// TIA Portal project "VISU_Registerlager_Template" (V14)

(* hardware
DEVICE "S7300/ET200M-Station_1"  S7-300 station
   slot 0: "Profilschiene_0"  Rail  6ES7 390-1***0-0AA0
   slot 2: "PLC_1"  CPU 315-2 PN/DP  6ES7 315-2EH13-0AB0  V2.6
      slot 1: "MPI/DP-Schnittstelle_1"  X1
      slot 2: "PROFINET-Schnittstelle_1"  PN-IO
         slot 1: "Port_1"  Port
*)

// ===== PLC "PLC_1"  CPU 315-2 PN/DP =====

VAR_GLOBAL   // PLC tag table "Standard-Variablentabelle"
   "CHAIN_REGISTER" AT %I10.0 : Bool;   // Förderkette Registerlager
   "REGISTER_ENGAGED" AT %I10.1 : Bool;   // Registerlager belegt
   "BELT_ENGAGED" AT %I10.2 : Bool;   // Förderband belegt
   "READ_SENSOR1" AT %I10.3 : Bool;   // Lesestation Sensor 1
   "READ_SENSOR2" AT %I10.4 : Bool;   // Lesestation Sensor 2
   "CONTROL_KEY" AT %I10.5 : Bool;   // Bedientaster
   "CHAIN_ON" AT %Q4.0 : Bool;   // Förderkette Regtisterlager an
   "LED_ON" AT %Q4.2 : Bool;   // LED an
   "BOX_NO" AT %MD1000 : DInt;   // Box-Nummer
   "BELT_ON" AT %Q4.1 : Bool;   // Förderband an
   "Merker TOF aktiv" AT %M0.0 : Bool;
   "Tag_4" AT %M0.5 : Bool;
   "Tag_3" AT %M0.4 : Bool;
   "Merker, 15 sec timer done" AT %M0.1 : Bool;
   "BOX_COUNTER1" AT %MW6 : Int;
   "BOX_COUNTER2" AT %MW8 : Int;
   "Tag_2" AT %M0.3 : Bool;
   "Tag_1" AT %M0.2 : Bool;
END_VAR

ORGANIZATION_BLOCK "Main"   // OB1, FBD
TITLE = "Main Program Sweep (Cycle)"
{ S7_Optimized_Access := 'FALSE' }
VERSION : 0.1
   VAR_TEMP
      OB1_EV_CLASS : Byte;   // Bits 0-3 = 1 (Coming event), Bits 4-7 = 1 (Event class 1)
      OB1_SCAN_1 : Byte;   // 1 (Cold restart scan 1 of OB 1), 3 (Scan 2-n of OB 1)
      OB1_PRIORITY : Byte;   // Priority of OB Execution
      OB1_OB_NUMBR : Byte;   // 1 (Organization block 1, OB1)
      OB1_RESERVED_1 : Byte;   // Reserved for system
      OB1_RESERVED_2 : Byte;   // Reserved for system
      OB1_PREV_CYCLE : Int;   // Cycle time of previous OB1 scan (milliseconds)
      OB1_MIN_CYCLE : Int;   // Minimum cycle time of OB1 (milliseconds)
      OB1_MAX_CYCLE : Int;   // Maximum cycle time of OB1 (milliseconds)
      OB1_DATE_TIME : Date_And_Time;   // Date and time OB1 started
   END_VAR
   VAR_TEMP   // added for the SCL form of the ladder/FBD networks
      _w1 : Bool;
      _w2 : Bool;
   END_VAR
BEGIN

REGION Network 1: Förderband an
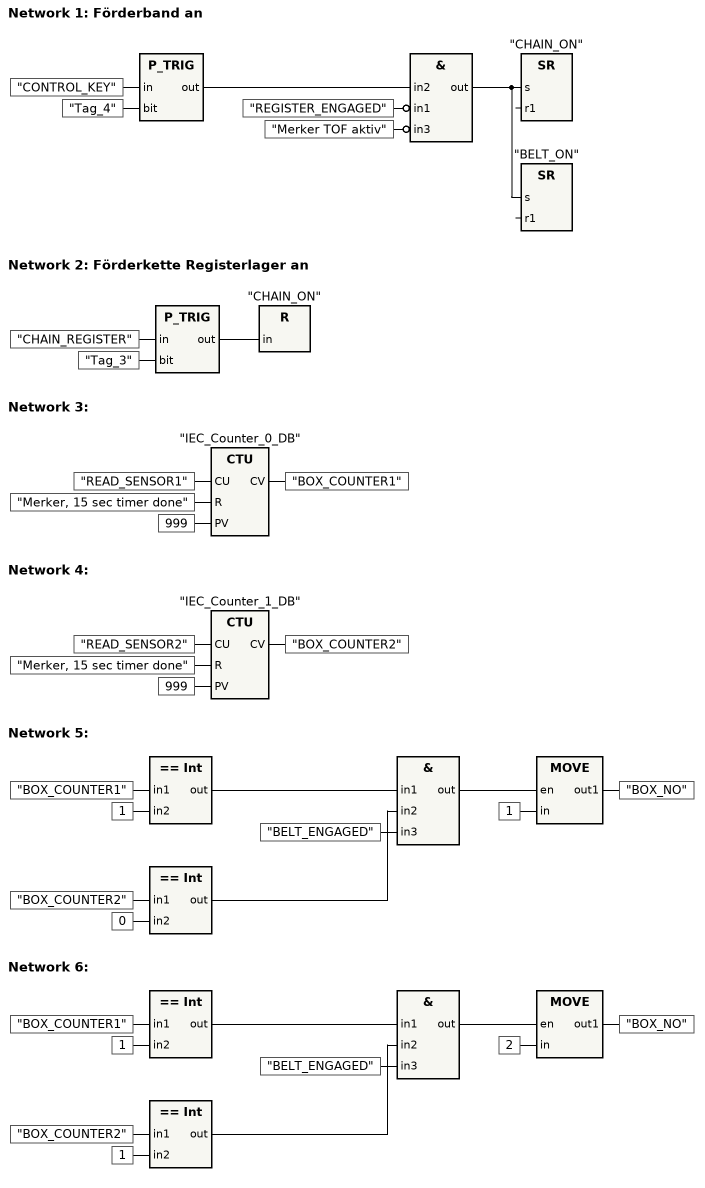
   #_w1 := "CONTROL_KEY" AND NOT "Tag_4";   // rising edge
   "Tag_4" := "CONTROL_KEY";
   #_w2 := #_w1 AND NOT "REGISTER_ENGAGED" AND NOT "Merker TOF aktiv";
   IF #_w2 THEN
       "CHAIN_ON" := TRUE;   // SR flip-flop
       "BELT_ON" := TRUE;   // SR flip-flop
   END_IF;
END_REGION

REGION Network 2: Förderkette Registerlager an
   #_w1 := "CHAIN_REGISTER" AND NOT "Tag_3";   // rising edge
   "Tag_3" := "CHAIN_REGISTER";
   IF #_w1 THEN "CHAIN_ON" := FALSE; END_IF;
END_REGION

REGION Network 3
   "IEC_Counter_0_DB".CTU(CU := "READ_SENSOR1",
                          R := "Merker, 15 sec timer done",
                          PV := 999,
                          CV => "BOX_COUNTER1");
END_REGION

REGION Network 4
   "IEC_Counter_1_DB".CTU(CU := "READ_SENSOR2",
                          R := "Merker, 15 sec timer done",
                          PV := 999,
                          CV => "BOX_COUNTER2");
END_REGION

REGION Network 5
   IF ("BOX_COUNTER1" = 1) AND ("BOX_COUNTER2" = 0) AND "BELT_ENGAGED" THEN "BOX_NO" := 1; END_IF;
END_REGION

REGION Network 6
   IF ("BOX_COUNTER1" = 1) AND ("BOX_COUNTER2" = 1) AND "BELT_ENGAGED" THEN "BOX_NO" := 2; END_IF;
END_REGION

REGION Network 7
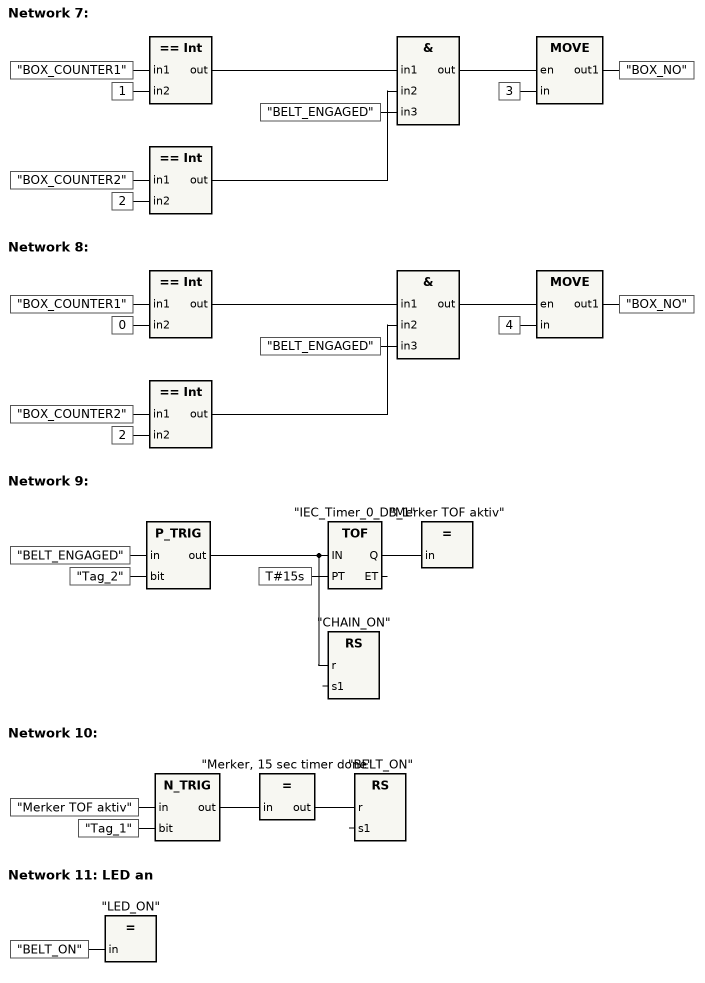
   IF ("BOX_COUNTER1" = 1) AND ("BOX_COUNTER2" = 2) AND "BELT_ENGAGED" THEN "BOX_NO" := 3; END_IF;
END_REGION

REGION Network 8
   IF ("BOX_COUNTER1" = 0) AND ("BOX_COUNTER2" = 2) AND "BELT_ENGAGED" THEN "BOX_NO" := 4; END_IF;
END_REGION

REGION Network 9
   #_w1 := "BELT_ENGAGED" AND NOT "Tag_2";   // rising edge
   "Tag_2" := "BELT_ENGAGED";
   "IEC_Timer_0_DB_1".TOF(IN := #_w1, PT := T#15s);
   "Merker TOF aktiv" := "IEC_Timer_0_DB_1".Q;
   IF #_w1 THEN
       "CHAIN_ON" := FALSE;   // RS flip-flop
   END_IF;
END_REGION

REGION Network 10
   #_w1 := NOT "Merker TOF aktiv" AND "Tag_1";   // falling edge
   "Tag_1" := "Merker TOF aktiv";
   "Merker, 15 sec timer done" := #_w1;
   IF #_w1 THEN
       "BELT_ON" := FALSE;   // RS flip-flop
   END_IF;
END_REGION

REGION Network 11: LED an
   "LED_ON" := "BELT_ON";
END_REGION
END_ORGANIZATION_BLOCK